FUNCTION ASIND : LREAL
VAR_INPUT
	SINVAL:LREAL;
END_VAR
VAR
END_VAR

ASIND:=RAD_TO_DEG(ASIN(SINVAL));

END_FUNCTION

(* stored: Version 1.1.0.1, ProductVersion 3.1.4024.12
   POU ASIND: Id {da8c1dfe-65c7-4b94-bf56-5cc6b8382315}, SpecialFunc None *)
